TYPE ST_Report :
STRUCT
	bStartCreate_Sequence				:BOOL;
	bStartSend_Sequence					:BOOL;
	bSend_Report						:BOOL;
	bExport_Alarms						:BOOL;
	bSaveAs_Alarms						:BOOL;
	bCreate_Report						:BOOL;
	bDelete_Data						:BOOL;
	bDelete_OldestReport				:BOOL;
END_STRUCT
END_TYPE

(* stored: Version 1.1.0.1, ProductVersion 3.1.4024.12
   DUT ST_Report: Id {1fa25576-b54b-4294-845c-8ae69b8846ff} *)
